Yaskawa INFORM job: CLEACING-STATION-2.JBI

/JOB
//NAME CLEACING-STATION-2
//POS
///NPOS 0,0,0,0,0,2
///TOOL 0
///POSTYPE ANGLE
///ANGLE
EX00040=180.0000
EX00041=-1.0000
//INST
///DATE 2018/10/02 11:29
///ATTR SC,RW
///GROUP1 ST2
NOP
SETE EX040 (1) 10000
SETE EX041 (1) -10000
*turn
IFTHEN IN#(19)=ON
	 IMOV EX040 VJ=25.00
ENDIF
IFTHEN IN#(20)=ON
	 IMOV EX041 VJ=25.00
ENDIF
JUMP *turn IF IN#(630)=OFF
END
